TYPE ST_Euchner_MGB2_HW_OUT :
STRUCT
	///Hardware Out
	nByte0: USINT;
END_STRUCT
END_TYPE

(* stored: Version 1.1.0.1, ProductVersion 3.1.4024.12
   DUT ST_Euchner_MGB2_HW_OUT: Id {6f4ec8dd-4db3-44b0-a479-2d1a76085304} *)
